TYPE ST_AmrModule_HMI :
	STRUCT
		Override : LREAL := 100.0;
	END_STRUCT
END_TYPE

(* stored: Version 1.1.0.1
   DUT ST_AmrModule_HMI: Id {6373cca3-230c-4786-9bdb-9be1cdb0f308} *)
